FUNCTION_BLOCK FB_SelfTest EXTENDS FB_StateMachine IMPLEMENTS I_StateMachine
VAR_INPUT
	bStart : BOOL;
	fbStepper : REFERENCE TO FB_Stepper;
	fbLinearActuator : REFERENCE TO FB_LinearActuator;
	fbJointSR : REFERENCE TO FB_Joint;
END_VAR
VAR_OUTPUT
END_VAR
VAR
	eInnerState : E_SelftestStates;
	bCompleted : BOOL;
	dtTimeCompleted: DATE_AND_TIME;
END_VAR

OuterLopSM();

METHOD Disable : BOOL

VAR
	bChildBusy  : BOOL := FALSE;
END_VAR
fbStepper.Active:=FALSE;
fbLinearActuator.Active:=FALSE;
fbJointSR.Active:=FALSE;

Disable := TRUE;
END_METHOD

METHOD InnerLoopSM : BOOL
// update all children FBs
// call to fbStepper() done by the parent (FB_ControllerArm) 

CASE CyclicInnerCase(TO_STRING(eInnerState)) OF
	E_SelftestStates.Idle:
		IF bStart THEN
			bStart := FALSE;
			ChangeInnerState(E_SelftestStates.HomeStepper1);
		END_IF
	
	E_SelftestStates.HomeStepper1:
		IF fbStepper.Busy THEN
			// fbStepper should never be busy here 	
			sErrorDetails := 'fbStepper.Busy = TRUE';
			fbEventHandler(eNapID:=E_Event.UNABLE_TO_START_TASK,sMessage:=sErrorDetails);
			bError := TRUE;
		ELSE	
			IF fbStepper.bError THEN
				sErrorDetails := 'fbStepper.bReady=FALSE';
				fbEventHandler(eNapID:=E_Event.UNABLE_TO_START_TASK,sMessage:=sErrorDetails);
				bError := TRUE;
			ELSE
				fbStepper.bStartHoming:=TRUE;
				ChangeInnerState(E_SelftestStates.HomeStepper2);
			END_IF
		END_IF


	E_SelftestStates.HomeStepper2:
		IF fbStepper.Busy THEN
			// Wait... fbStepper still busy 	
		ELSE
			IF fbStepper.bError THEN
				fbEventHandler(eNapID:=E_Event.TASK_FAILED,sTrace:=fbStepper.EventTrace);
				fbStepper.ErrorAck:=TRUE;
				bError := TRUE;
			ELSE
				IF fbStepper.Homed THEN
					ChangeInnerState(E_SelftestStates.HomeLinearActuator1);
				ELSE
					sErrorDetails := 'fbStepper.Homed=FALSE';
					fbEventHandler(eNapID:=E_Event.TASK_FAILED,sMessage:=sErrorDetails);
					bError := TRUE;
				END_IF
			END_IF
		END_IF
		
	E_SelftestStates.HomeLinearActuator1:
		IF fbLinearActuator.Busy THEN
			// fbStepper should never be busy here 	
			sErrorDetails := 'fbLinearActuator.Busy = TRUE';
			fbEventHandler(eNapID:=E_Event.UNABLE_TO_START_TASK,sMessage:=sErrorDetails);
			bError := TRUE;
		ELSE	
			IF fbLinearActuator.bError THEN
				sErrorDetails := 'fbLinearActuator.bReady=FALSE';
				fbEventHandler(eNapID:=E_Event.UNABLE_TO_START_TASK,sMessage:=sErrorDetails);
				bError := TRUE;
			ELSE
				fbLinearActuator.bStartHoming:=TRUE;
				ChangeInnerState(E_SelftestStates.HomeLinearActuator2);
			END_IF
		END_IF
		
	E_SelftestStates.HomeLinearActuator2:
		IF fbLinearActuator.Busy THEN
			// Wait... fbLinearActuator still busy 	
		ELSE
			IF fbLinearActuator.bError THEN
				fbEventHandler(eNapID:=E_Event.TASK_FAILED,sTrace:=fbLinearActuator.EventTrace);
				fbLinearActuator.ErrorAck:=TRUE;
				bError := TRUE;
			ELSE
				IF fbLinearActuator.Homed THEN
					ChangeInnerState(E_SelftestStates.SetupEncoders1);
				ELSE
					sErrorDetails := 'fbLinearActuator.Homed=FALSE';
					fbEventHandler(eNapID:=E_Event.TASK_FAILED,sMessage:=sErrorDetails);
					bError := TRUE;
				END_IF
			END_IF
		END_IF
	
	E_SelftestStates.SetupEncoders1:
		IF fbJointSR.Busy THEN
			// fbJointSR should never be busy here 	
			sErrorDetails := 'fbJointSR.Busy = TRUE';
			fbEventHandler(eNapID:=E_Event.UNABLE_TO_START_TASK,sMessage:=sErrorDetails);
			bError := TRUE;
		ELSE	
			IF fbJointSR.bError THEN
				sErrorDetails := 'fbJointSR.bReady=FALSE';
				fbEventHandler(eNapID:=E_Event.UNABLE_TO_START_TASK,sMessage:=sErrorDetails);
				bError := TRUE;
			ELSE
				fbJointSR.bStartSetup:=TRUE;
				ChangeInnerState(E_SelftestStates.SetupEncoders2);
			END_IF
		END_IF
		
	E_SelftestStates.SetupEncoders2:
		IF fbJointSR.Busy THEN
			// Wait... fbJointSR still busy 	
		ELSE
			IF fbJointSR.bError THEN
				fbEventHandler(eNapID:=E_Event.TASK_FAILED,sTrace:=fbLinearActuator.EventTrace);
				fbLinearActuator.ErrorAck:=TRUE;
				bError := TRUE;
			ELSE
				IF fbJointSR.Calibrated THEN
					ChangeInnerState(E_SelftestStates.CheckAbsEncoderOffsets1);
				ELSE
					sErrorDetails := 'fbLinearActuator.Homed=FALSE';
					fbEventHandler(eNapID:=E_Event.TASK_FAILED,sMessage:=sErrorDetails);
					bError := TRUE;
				END_IF
			END_IF
		END_IF
		
	E_SelftestStates.CheckAbsEncoderOffsets1:
		ChangeInnerState(E_SelftestStates.CheckAbsEncoderOffsets2);
		
	E_SelftestStates.CheckAbsEncoderOffsets2:
		ChangeInnerState(E_SelftestStates.WrapUp);
		
	E_SelftestStates.WrapUp:
		bCompleted := TRUE;
		dtTimeCompleted := DateTime.GVL_DATE_TIME;
		fbEventHandler(eNapID:=E_Event.REQUEST_COMPLETED);
		ChangeInnerState(E_SelftestStates.Idle);
END_CASE
END_METHOD

METHOD Reset : BOOL
// reset variables specific to this FB 
bCompleted := FALSE;
dtTimeCompleted := DATE_AND_TIME#1970-1-1-0:0:0;
END_METHOD

PROPERTY SelftestNeeded : BOOL
GET
// TODO: Check if dtTimeCompleted is too old. If so set SelftestNeeded := TRUE
SelftestNeeded := NOT bCompleted;
END_GET
END_PROPERTY

METHOD Setup : BOOL
eStateMachineSourceID := eStateSourceID;
SetInnerEnumeration(nStateEnum:=THIS^.eInnerState);
END_METHOD

PROPERTY TimeCompleted : DATE_AND_TIME
GET
TimeCompleted := dtTimeCompleted;
END_GET
END_PROPERTY

END_FUNCTION_BLOCK

(* stored: Version 1.1.0.1, ProductVersion 3.1.4024.12
   POU FB_SelfTest: Id {1bb06a1d-0466-4467-bee4-d88d42712776}, SpecialFunc None
   Folder Properties: Id {b682ec8a-b81c-4636-afdb-e735070caa7e}
   Method Disable: Id {24cb7115-e443-47a2-b5bf-65e04415eec9}
   Method InnerLoopSM: Id {1533b789-f1f5-4dea-814a-7ae4a8c15ba7}
   Method Reset: Id {0271353f-d7b7-4a53-aa67-eed09f291c10}
   Property SelftestNeeded: Id {057e6406-8538-41aa-9d0c-3467e2ddc63d}
   Get Get: Id {747024a2-f3ae-4631-b586-35e134748b51}
   Method Setup: Id {fdd0c095-c587-4815-b66b-4d1d74983531}
   Property TimeCompleted: Id {1cbfd24b-c535-454b-97a1-c0e9fffacf40}
   Get Get: Id {f251df04-d6e9-40c1-9b07-1613530dd50c} *)
